// Base class of modules with axis and buttons for manual control
FUNCTION_BLOCK FB_Subsystem_Root
VAR_INPUT	
	// =============== Axis button variables =====================
	bButtonAxisFwIn				: BOOL;						// Signal of button to move axis forwards
	bButtonAxisBwIn				: BOOL;						// Signal of button to move axis backwards
END_VAR
VAR_OUTPUT
	// =============== Error variables ===========================
	bAxisError					: BOOL;						// Error signal of axis
	nAxisErrorID				: UDINT;					// Error ID of axis error

	// =============== Axis, button and module return signals ====
	bAxisMoves					: BOOL;						// True if axis is moving
	bButtonAxisFwOut			: BOOL;						// Processed signal for button to move axis forwards
	bButtonAxisBwOut			: BOOL;						// Processed signal for button to move axis backwards			
END_VAR
VAR
	// =============== Done signals of Halt, Reset and Starting ==
	bHaltDone					: BOOL;						// True if module is stopped
	bResetDone					: BOOL;						// True if module is reset
	bStartingDone				: BOOL;						// True if module is started
	
	// =============== Enables ===================================
	bComprAirEnabledLocal		: BOOL;						// Enable of compressed air
	bAxisEnableLocal			: BOOL;						// Enable of axis
	bSensorEnableLocal			: BOOL;						// Enable of sensor
	bManualAxisEnableLocal		: BOOL;						// Enable of manual axis control
	bManualCylinderEnable		: BOOL;						// Enable of manual cylinder control (not written with input of method Enable)

	// =============== State variables ===========================
	bHaltRequest				: BOOL;						// True if machine is in state ABORTING or STOPPING
	bResetRequest				: BOOL;						// True if machine is in state RESETTING

	// =============== Axis ======================================
	fbAxis						: FB_Axis;					// Function block instance of FB_Axis
	fAxisVelo					: LREAL;					// Velocity of axis
	
	// =============== Manual axis control =======================
	fbButtonAxisFw				: FB_SignalHandlingIntern;	// To move axis forwards	
	fbButtonAxisBw				: FB_SignalHandlingIntern;	// To move axis backwards
	
	// =============== Common variables ==========================
	fbTriggerStartingStart		: R_TRIG;					// To diagnose rising edge of starting action starting
	fbTriggerResetStart			: R_TRIG;					// To diagnose rising edge of starting reset			
	bMoved						: BOOL;						// History variable to save if axis has moved
END_VAR

// =========================================================
;
// =========================================================

PROPERTY bState_HaltDone : BOOL
GET
bState_HaltDone := bHaltDone;
END_GET
END_PROPERTY

PROPERTY bState_ResetDone : BOOL
GET
bState_ResetDone := bResetDone;
END_GET
END_PROPERTY

PROPERTY bState_StartingDone : BOOL
GET
bState_StartingDone := bStartingDone;
END_GET
END_PROPERTY

METHOD PUBLIC Enable
VAR_INPUT
	bComprAirEnabled		: BOOL;			// Enable of compressed air
	bAxisEnable				: BOOL;			// Enable of axis
	bSensorEnable			: BOOL;			// Enable of sensor
	bManualAxisEnable		: BOOL;			// Enable of manual axis control
END_VAR
// =========================================================
// Store inputs in local variables

	bComprAirEnabledLocal	:= bComprAirEnabled;
	bAxisEnableLocal		:= bAxisEnable;
	bSensorEnableLocal		:= bSensorEnable;
	bManualAxisEnableLocal	:= bManualAxisEnable;
	
// =========================================================	
// Enable axis

	fbAxis.Enable(bEnable := bAxisEnableLocal);					

// =========================================================
// Enable cylinder
		
	bManualCylinderEnable := bManualAxisEnableLocal AND bComprAirEnabledLocal;

// =========================================================
// Control of axis button
		
	fbButtonAxisFw.Enable(bEnable := bManualAxisEnableLocal AND NOT fbButtonAxisBw.bOut);
	fbButtonAxisBw.Enable(bEnable := bManualAxisEnableLocal AND NOT fbButtonAxisFw.bOut);

// =========================================================
END_METHOD

PROPERTY fAxisVelocity : LREAL
GET
fAxisVelocity := fAxisVelo;
END_GET
SET
fAxisVelo := fAxisVelocity;
END_SET
END_PROPERTY

METHOD PUBLIC Halt
VAR_INPUT
	bHalt		: BOOL;				// True if machine is in state ABORTING or STOPPING
END_VAR
// =========================================================
// Store request

	bHaltRequest := bHalt;

// =========================================================
// Halting axis

	fbAxis.Halt(bDriveHalt := bHaltRequest);

// =========================================================
// Getting halt state

	bHaltDone := fbAxis.bState_HaltDone;

// =========================================================
END_METHOD

METHOD PUBLIC InputOutput
VAR_INPUT
END_VAR
// =========================================================
// Axis buttons and output variable for axis
		
	fbButtonAxisFw.SetOutput();	
	fbButtonAxisBw.SetOutput();
	
	bAxisMoves 		:= fbAxis.bMoves;
	bAxisError		:= fbAxis.bError;
	nAxisErrorID	:= fbAxis.nErrorID;
	
	fbButtonAxisFw.bInput 	:= bButtonAxisFwIn;
	fbButtonAxisBw.bInput	:= bButtonAxisBwIn;
	bButtonAxisFwOut 		:= fbButtonAxisFw.bOut;
	bButtonAxisBwOut		:= fbButtonAxisBw.bOut;

// =========================================================
END_METHOD

METHOD PUBLIC Manual
VAR_INPUT
END_VAR
// =========================================================
// Manual axis control
	
	// Button to move axis backwards pressed
	IF fbButtonAxisBw.bOut THEN
		IF bHaltDone THEN
			bHaltDone := FALSE;
		END_IF
		
		IF NOT bMoved THEN
			bMoved := TRUE;
		END_IF
		
		// Move axis backwards
		fbAxis.MoveBw();
	
	// Button to move axis forwards pressed
	ELSIF fbButtonAxisFw.bOut THEN
		IF bHaltDone THEN
			bHaltDone := FALSE;
		END_IF
		
		IF NOT bMoved THEN
			bMoved := TRUE;
		END_IF
		
		// Move axis forwards
		fbAxis.MoveFw();
		
	// No button is pressed and halt is not done
	ELSIF NOT bHaltDone THEN
		// Request halt if axis has moved
		IF bMoved THEN
			Halt(bHalt := TRUE);
		END_IF
		
	// Halt is done but still requested
	ELSIF bHaltRequest THEN
		Halt(bHalt := FALSE);
		
		bMoved := FALSE;
	END_IF

// =========================================================
END_METHOD

METHOD PUBLIC Reset
VAR_INPUT
	bReset		: BOOL;				// True if machine is in state RESETTING
END_VAR
// =========================================================
// Store request

	bResetRequest := bReset;
	
// =========================================================
// Resetting variables

	bMoved 			:= FALSE;
	bHaltDone 		:= FALSE;
	bHaltRequest	:= FALSE;

// =========================================================
// Resetting axis
						
	fbTriggerResetStart(CLK := bReset);
	
	fbAxis.Reset(bDriveReset := bReset);
	
	bResetDone := fbAxis.bState_ResetDone;

// =========================================================
END_METHOD

METHOD PROTECTED ResetState
VAR_INPUT
END_VAR
// =========================================================
// Placeholder method for sub classes
;

// =========================================================
END_METHOD

METHOD PUBLIC Starting
VAR_INPUT
	bStarting		: BOOL;			// True if machine is in state STARTING
END_VAR
// =========================================================

fbTriggerStartingStart(CLK := bStarting);

IF fbTriggerStartingStart.Q THEN
	bStartingDone 			:= FALSE;
	// Setting velocity of axis
	fbAxis.fTargetVelocity 	:= fAxisVelo;
	// Resetting state variable
	ResetState();
END_IF

IF fbAxis.bState_Enable THEN
	bStartingDone := TRUE;
END_IF

// =========================================================
END_METHOD

METHOD PUBLIC Stop
VAR_INPUT
	bHalt		: BOOL;				// True if machine is in state ABORTING or STOPPING
END_VAR
// =========================================================
// Store request

	bHaltRequest := bHalt;

// =========================================================
// Stopping axis

	fbAxis.Stop(bDriveStop := bHaltRequest);
		
// =========================================================			
// Getting halt state

	bHaltDone := fbAxis.bState_HaltDone;

// =========================================================
END_METHOD

END_FUNCTION_BLOCK

(* stored: Version 1.1.0.1, ProductVersion 3.1.4024.2
   POU FB_Subsystem_Root: Id {029c4fe0-4583-4c3e-b473-0d6014ef191e}, SpecialFunc None
   Property bState_HaltDone: Id {51d4aac7-515c-43ce-a636-d67222abcbee}
   Get Get: Id {05dbbb6b-fefa-4bea-abd7-e4e89a196951}
   Property bState_ResetDone: Id {46ad43b2-b742-4219-8c98-95328ac55c23}
   Get Get: Id {8cef0182-e3ad-47ea-b311-5fef88266aa1}
   Property bState_StartingDone: Id {61ede4c9-887c-40c2-a81c-7bc94ab0ab02}
   Get Get: Id {fbd5058c-d215-4996-8e50-673191e29deb}
   Method Enable: Id {43c9b96b-8e65-42ff-abd4-fbf959f70451}
   Property fAxisVelocity: Id {4d3082cd-259a-469e-9cc6-05ec58b47804}
   Get Get: Id {738e152c-05d7-4318-a5f5-a55d14efb5da}
   Set Set: Id {9d5a6b82-eab7-4120-ba7d-8a6489e5a400}
   Method Halt: Id {700e424d-b225-4235-9098-b1ad26ce2872}
   Method InputOutput: Id {e67657ad-563d-4030-9632-361703757d9b}
   Method Manual: Id {e44b5b94-2008-45ac-af61-e442cb95047e}
   Method Reset: Id {61c05617-304d-4b33-aeda-05edbc2e76f6}
   Method ResetState: Id {dc0cb0f5-f280-4519-a21c-d84b6f8c68b4}
   Method Starting: Id {ac60b6b3-698c-4d83-9705-d6cc549cb6b2}
   Method Stop: Id {a6d8b6ed-ce1f-4cb9-a9fe-bbdf818e5733} *)
